//==================================================================================================
//								RJM Maszyny sp. z o.o.
//									13.05.2022
//	Obsługa silonwika z zawrorem 5 na 3 - Odpowietrzony
//	Realizacja wysuwania i chowania tłoczyska dla jednej cewki zwrócenie pozycji skrajnych
// 	v1.0	|| TC v 3.1.4024.22		|| - pierwsza wersja
//==================================================================================================
FUNCTION_BLOCK FB_Silownik_5na3_Odpowietrzony_Kontrola EXTENDS FB_SilownikBaza_Kontola
VAR_INPUT
END_VAR
VAR_OUTPUT
END_VAR
VAR
	bCewkaB							AT %Q*	: BOOL;	
END_VAR

METHOD Praca : BOOL
VAR_INPUT
END_VAR
SUPER^.Praca ();

IF (bPrzesuwanieWStroneKonca AND NOT bCewkaA) THEN
	bCewkaA									:= TRUE;
END_IF
IF  (bPrzesuwanieWStronePoczatku AND bCewkaA) THEN
	bCewkaA									:= FALSE;
END_IF

IF (bPrzesuwanieWStronePoczatku AND NOT bCewkaB) THEN
	bCewkaB									:= TRUE;
END_IF
IF  (bPrzesuwanieWStroneKonca AND bCewkaB) THEN
	bCewkaB									:= FALSE;
END_IF
END_METHOD

END_FUNCTION_BLOCK

(* stored: Version 1.1.0.1, ProductVersion 3.1.4024.11
   POU FB_Silownik_5na3_Odpowietrzony_Kontrola: Id {60dff856-85f7-4c6d-b839-86288f7fcaaa}, SpecialFunc None
   Method Praca: Id {01a46643-75e1-497b-a08a-28bc141dd980} *)
